KUKA KRL program: art_dispenser.src, art_dispenser.dat

--- art_dispenser.src ---
&ACCESS RVO2
&REL 380
&PARAM EDITMASK = *
&PARAM TEMPLATE = C:\KRC\Roboter\Template\vorgabe
&PARAM DISKPATH = KRC:\R1\TP\ART
DEF art_dispenser( )
END
;
;
;
GLOBAL DEF ARTDispenserInit()
   ART_dispenser[1].ready_error = FALSE
   ARTHMIClearMessage(ART_dispenser[1].m_disp_not_ready)
   ARTHMIClearMessage(ART_dispenser[1].m_disp_alarm)
   ARTHMIClearMessage(ART_dispenser[1].m_disp_low_level)
END
;
;
;
GLOBAL DEFFCT BOOL ARTDispencerGive()
   IF ART_dispenser[1].di_ready THEN
      ART_dispenser[1].do_request = TRUE
      RETURN TRUE
   ELSE
      ART_dispenser[1].ready_error = TRUE
      RETURN FALSE
   ENDIF
ENDFCT
;
;
;
GLOBAL DEF ARTDispenserConfirm()
   ART_dispenser[1].do_taken = TRUE
END
; **** SET GRIPPER TO THE INITIAL STATE
;
;
GLOBAL DEF ARTDispencerDoSPS()
   ;vars bind
   doDispenserRequest = ART_dispenser[1].do_request
   doDispenserTaken = ART_dispenser[1].do_taken

   ART_dispenser[1].di_ready = diDispenserReady
   ART_dispenser[1].di_ready_take =  diDispenserReadyTake
   ART_dispenser[1].di_alarm = diDispenserAlarm
   ART_dispenser[1].di_low_level = diDispenserLow

   IF ARTHMIIsResetPushed() THEN
      ART_dispenser[1].ready_error = FALSE
      ARTHMIClearMessage(ART_dispenser[1].m_disp_not_ready)
      ARTHMIClearMessage(ART_dispenser[1].m_disp_alarm)
      ARTHMIClearMessage(ART_dispenser[1].m_disp_low_level)
      ART_dispenser[1].error_state = #NORMAL
   ENDIF
   ; Swith off Request signal
   IF ART_dispenser[1].di_ready_take THEN
      ART_dispenser[1].do_request = FALSE
   ENDIF
   ; Swith off Taken signal
   IF ART_dispenser[1].di_ready THEN
      ART_dispenser[1].do_taken = FALSE
   ENDIF
   ; Errors
   IF ART_dispenser[1].di_alarm THEN
      ARTHMISetMessage(ART_dispenser[1].m_disp_alarm,TRUE,"ARTDispenser", "DISPENSER_ALARM")
      ARTSystemSetState(#ARTSYS_STATE_WARNING)
      ART_dispenser[1].error_state = #ERROR
   ENDIF

   IF ART_dispenser[1].di_low_level THEN
      ARTHMISetMessage(ART_dispenser[1].m_disp_low_level,TRUE,"ARTDispenser", "DISPENSER_LOW_LEVEL")
      ARTSystemSetState(#ARTSYS_STATE_WARNING)
      ART_dispenser[1].error_state = #WARNING
   ENDIF

   IF ART_dispenser[1].ready_error THEN
      ARTHMISetMessage(ART_dispenser[1].m_disp_not_ready,TRUE,"ARTDispenser", "DISPENSER_NOT_READY")
      ARTSystemSetState(#ARTSYS_STATE_WARNING)
      ART_dispenser[1].error_state = #ERROR
   ENDIF
   ; test
   IF doTestGivePallet THEN
      IF ARTDispencerGive() THEN
         doTestGivePallet = FALSE
      ENDIF
   ENDIF
END

--- art_dispenser.dat ---
&ACCESS RVO2
&REL 380
&PARAM EDITMASK = *
&PARAM TEMPLATE = C:\KRC\Roboter\Template\vorgabe
&PARAM DISKPATH = KRC:\R1\TP\ART
DEFDAT  art_dispenser PUBLIC
   GLOBAL STRUC DISPENCER ART_DEVICE_STATE error_state, BOOL ready_error,BOOL do_request,BOOL do_taken,BOOL di_ready,BOOL di_ready_take,BOOL di_alarm,BOOL di_low_level,INT m_disp_not_ready, INT m_disp_alarm, INT m_disp_low_level
   DECL GLOBAL DISPENCER ART_dispenser[1]
   ART_dispenser[1] = {error_state #NORMAL, ready_error FALSE,do_request FALSE,do_taken FALSE,di_ready FALSE,di_ready_take FALSE,di_alarm FALSE,di_low_level FALSE,m_disp_not_ready 0,m_disp_alarm 0,m_disp_low_level 0}
ENDDAT
